# EPICS autosave request: BPMApp/Db/BPMInfo_settings.req
# Nothing needs to be saved here
$(P)$(R)INFOHarmonicNumber
$(P)$(R)INFOClkFreq
$(P)$(R)INFOClkProp
$(P)$(R)INFOTBTRate
$(P)$(R)INFOFOFBRate
$(P)$(R)INFOMONITRate
